{attribute 'GeneratedUsingTerminal: EJ1914-0000-0017'}
{attribute addProperty BoxType "EJ1914-0000-0017"}
{attribute addProperty Id "Module_1_FSOEModule_1_FSOE_5515F18A18Module_2_DEVICEIOModule_2_DEVICEIO_5FA6B4E72Module_3_FSLOGICModule_3_FSLOGIC_DEAB45222WcStateAT %I*WcState_9091E0EB2InfoDataAT %I*InfoData_94A18F5E2"}
{attribute addProperty CRC "2175977418"}
{attribute addProperty Size "26"}
TYPE EJ1914_81B2C7CA EXTENDS EtcSlaveTerminalBase_947E5A46 :
STRUCT
	{attribute addProperty Name "Module_1_FSOE"}
	Module_1_FSOE : Module_1_FSOE_5515F18A;
	{attribute addProperty Name "Module_2_DEVICEIO"}
	Module_2_DEVICEIO : Module_2_DEVICEIO_5FA6B4E7;
	{attribute addProperty Name "Module_3_FSLOGIC"}
	Module_3_FSLOGIC : Module_3_FSLOGIC_DEAB4522;
	{attribute addProperty Name "WcState"}
	WcState : WcState_9091E0EB;
	{attribute addProperty Name "InfoData"}
	InfoData : InfoData_94A18F5E;
END_STRUCT
END_TYPE

(* stored: Version 1.2.0.0, ProductVersion 3.1.4024.9
   DUT EJ1914_81B2C7CA: Id {37db7360-1fc9-4b66-9712-817e0a2941cb} *)
